PROGRAM OPERATION_Controller
VAR	
	xHomeRunExecute:		BOOL;
	xDone:					BOOL;
	xHomeOK:				BOOL;
	
	rtControlOn:			R_TRIG;
	rtHomeRunDone:			R_TRIG;
	
	fbHOME_RUN:				HOME_RUN_SEQ;
END_VAR

rtControlOn(CLK:=G_xAutoMode);
rtHomeRunDone(CLK:=xDone);

IF rtControlOn.Q AND xHomeOK AND G_xPowerOn AND NOT G_xErrorExist THEN xHomeRunExecute:=TRUE; ELSE xHomeRunExecute:=FALSE; END_IF
IF rtHomeRunDone.Q THEN xHomeOK:=TRUE; END_IF

fbHOME_RUN(	xExecute:=xHomeRunExecute, xDone:=xDone);

//Szeretem az almaspitet''''

END_PROGRAM

(* stored: Version 1.1.0.1, ProductVersion 3.1.4022.18
   POU OPERATION_Controller: Id {2c77ea48-d508-49bc-a424-4f74a9e55231}, SpecialFunc None *)
